Yaskawa INFORM job: GRIP_2FG7-2.JBI

/JOB
//NAME GRIP_2FG7-2
//POS
///NPOS 0,0,0,0,0,0
//INST
///DATE 2023/11/30 18:20
///ATTR SC,RW
///GROUP1 RB1
NOP
CALL JOB:OR_INIT ARGF103 ARGF16
CALL JOB:OR_TWOFG_GRIP ARGF2 ARGF40 ARGF50 ARGF100 ARGF1
END
